(* CoDeSys 2.3.5.6 project: lyjak_02_st.pro *)
(* Author: mgr inż. Tomasz Sklenarski *)
(* Libraries: Standard.lib*4.1.15 17:23:13, SYSLIBCALLBACK.LIB*4.1.15 17:23:13 *)

(* PLC configuration (modules and I/O channels)
I1 AT %IX0.0 [LocalBitInput] Input I1
I2 AT %IX0.1 [LocalBitInput] Input I2
I3 AT %IX0.2 [LocalBitInput] Input I3
I4 AT %IX0.3 [LocalBitInput] Input I4
I5 AT %IX0.4 [LocalBitInput] Input I5
I6 AT %IX0.5 [LocalBitInput] Input I6
I7 AT %IX0.6 [LocalBitInput] Input I7
I8 AT %IX0.7 [LocalBitInput] Input I8
I9 AT %IX1.0 [LocalBitInput] Input I9
I10 AT %IX1.1 [LocalBitInput] Input I10
I11 AT %IX1.2 [LocalBitInput] Input I11
I12 AT %IX1.3 [LocalBitInput] Input I12
I13 AT %IX1.4 [LocalDiagInput] Diagnostic Input I13
I14 AT %IX1.5 [LocalDiagInput] Diagnostic Input I14
I15 AT %IX1.6 [LocalDiagInput] Diagnostic Input I15
I16 AT %IX1.7 [LocalDiagInput] Diagnostic Input I16
I7_Analog AT %IW2 [LocalAnalogIn] Input I7, 10Bit, 0-10VDC
I8_Analog AT %IW4 [LocalAnalogIn] Input I8, 10Bit, 0-10VDC
I11_Analog AT %IW6 [LocalAnalogIn] Input I11, 10Bit, 0-10VDC
I12_Analog AT %IW8 [LocalAnalogIn] Input I12, 10Bit, 0-10VDC
Q1 AT %QX0.0 [LocalBitOutput] Transistor-Output Q1
Q2 AT %QX0.1 [LocalBitOutput] Transistor-Output Q2
Q3 AT %QX0.2 [LocalBitOutput] Transistor-Output Q3
Q4 AT %QX0.3 [LocalBitOutput] Transistor-Output Q4
Q5 AT %QX0.4 [LocalBitOutput] Transistor-Output Q5
Q6 AT %QX0.5 [LocalBitOutput] Transistor-Output Q6
Q7 AT %QX0.6 [LocalBitOutput] Transistor-Output Q7
Q8 AT %QX0.7 [LocalBitOutput] Transistor-Output Q8
No Analog Output [EC4P_NoAnalogOutput] node 1, in %IB10 out %QB1
No Keys [EC4P_NoKeys] node 2, in %IB10 out %QB1
No Counter [EC4P_NoCounter] node 3, in %IB10 out %QB1
Extension [EC4P_Extension] node 1, in %IB10 out %QB1
  No Extension [EC4P_NoExtension] node 0, in %IB10 out %QB1
*)

(* Global variable list: ilosc_bitow_porownania *)
VAR_GLOBAL CONSTANT
	MaxNoOfStates: UINT:=26;
END_VAR

(* Global variable list: wizualizacja *)
VAR_GLOBAL
	numerStanuIn1:BYTE;
	numerStanuIn2:BYTE;
END_VAR

(* Global variable list: ZMIENNE_WYMIANY *)
VAR_GLOBAL
	sterowanieQ12:dataExchange;
	sterowanieQ34:dataExchange;
END_VAR

(* Data type *)
TYPE dataExchange :
STRUCT
	InputState:ARRAY[0..MaxNoOfStates]OF signal;
	Qa:ARRAY[0..MaxNoOfStates]OF signal;
	Qb:ARRAY[0..MaxNoOfStates]OF signal;
END_STRUCT
END_TYPE

(* Data type *)
TYPE signal: (e0, e1, eXX);
END_TYPE

(* POU PLC_PRG, ST *)
PROGRAM PLC_PRG
VAR

	firstRun:BOOL;
	scanner1: scan;
	scan1No:BYTE;
	scanner2: scan;
	scan2No:BYTE;
END_VAR
IF NOT firstRun THEN
i1_config;
i2_config;
firstRun:=TRUE;
END_IF
scanner1(DigIn:=I1 , sigDef:=ADR(sterowanieQ12) , QA=>Q1 , QB=>Q2, No=> numerStanuIn1 );
scanner2(DigIn:=I1 , sigDef:=ADR(sterowanieQ34) , QA=>Q3 , QB=>Q4, No=> numerStanuIn2);
END_PROGRAM
ACTION i1_config:
sterowanieQ12.InputState[2]:=e1;
sterowanieQ12.InputState[3]:=e1;
sterowanieQ12.InputState[4]:=e1;
sterowanieQ12.InputState[5]:=e1;
sterowanieQ12.InputState[6]:=e1;
sterowanieQ12.InputState[7]:=e1;
sterowanieQ12.InputState[8]:=e1;
sterowanieQ12.InputState[9]:=eXX;
sterowanieQ12.InputState[10]:=eXX;
sterowanieQ12.InputState[11]:=e1;
sterowanieQ12.InputState[12]:=e1;

sterowanieQ12.Qa[5]:=e1;
sterowanieQ12.Qa[6]:=e1;
sterowanieQ12.Qa[7]:=e1;
(*
sterowanieQ12.Qa[9]:=eXX;
sterowanieQ12.Qa[10]:=eXX;
*)
sterowanieQ12.Qa[14]:=e1;
sterowanieQ12.Qa[15]:=e1;
sterowanieQ12.Qa[16]:=e1;


sterowanieQ12.Qb[2]:=e1;
sterowanieQ12.Qb[3]:=e1;
sterowanieQ12.Qb[5]:=e1;
sterowanieQ12.Qb[6]:=e1;
(*
sterowanieQ12.Qb[9]:=eXX;
sterowanieQ12.Qb[10]:=eXX;
*)
sterowanieQ12.Qb[17]:=e1;
sterowanieQ12.Qb[18]:=e1;
sterowanieQ12.Qb[21]:=e1;
sterowanieQ12.Qb[22]:=e1;
END_ACTION
ACTION i2_config:
sterowanieQ34.InputState[2]:=e1;
sterowanieQ34.InputState[3]:=e1;
sterowanieQ34.InputState[4]:=e1;
sterowanieQ34.InputState[5]:=e1;
sterowanieQ34.InputState[6]:=e1;
sterowanieQ34.InputState[7]:=e1;
sterowanieQ34.InputState[8]:=e1;
sterowanieQ34.InputState[9]:=e1;
sterowanieQ34.InputState[10]:=e1;
sterowanieQ34.InputState[11]:=eXX;
sterowanieQ34.InputState[12]:=eXX;
sterowanieQ34.InputState[13]:=e1;
sterowanieQ34.InputState[14]:=e1;
sterowanieQ34.InputState[15]:=e1;
sterowanieQ34.InputState[16]:=e1;

sterowanieQ34.Qa[4]:=e1;
sterowanieQ34.Qa[5]:=e1;
sterowanieQ34.Qa[8]:=e1;
sterowanieQ34.Qa[9]:=e1;
sterowanieQ34.Qa[17]:=e1;
sterowanieQ34.Qa[18]:=e1;
sterowanieQ34.Qa[21]:=e1;
sterowanieQ34.Qa[22]:=e1;

sterowanieQ34.Qb[2]:=e1;
sterowanieQ34.Qb[3]:=e1;
sterowanieQ34.Qb[4]:=e1;
sterowanieQ34.Qb[19]:=e1;
sterowanieQ34.Qb[20]:=e1;
END_ACTION

(* POU scan, ST *)
FUNCTION_BLOCK scan
VAR_INPUT
	DigIn:BOOL;
	sigDef:POINTER TO dataExchange;
END_VAR
VAR_OUTPUT
	QA:BOOL;
	QB:BOOL;
	No:BYTE;
END_VAR
VAR
	tim: TON;
	StateMachine:BYTE;
	StateTime:TIME:=t#1s;
END_VAR
CASE StateMachine
OF
0:
IF DigIn THEN
REPEAT
No:=No+1;
UNTIL sigDef^.InputState[No]=e0
END_REPEAT
No:=No+1;
StateMachine:=1;
END_IF
1:
IF tim.Q THEN

IF NOT DigIn AND sigDef^.InputState[No]=eXX THEN
StateMachine:=2;
END_IF
END_IF
2:
StateTime:=t#2s;
IF tim.Q THEN
StateMachine:=3;
StateTime:=t#1s;
END_IF
3:
IF DigIn THEN
StateMachine:=1;
END_IF
END_CASE


tim(IN:=(StateMachine=1 OR StateMachine=2 OR StateMachine=4) AND NOT tim.Q , PT:=StateTime , Q=> , ET=> );
IF tim.Q THEN
No:=No+1;
END_IF
IF No>=MaxNoOfStates THEN
No:=UINT_TO_BYTE(MaxNoOfStates);
END_IF


QA:=sigToBOOL(sigDef^.Qa[No]);
QB:=sigToBOOL(sigDef^.Qb[No]);
END_FUNCTION_BLOCK

(* POU sigToBOOL, ST *)
FUNCTION sigToBOOL : BOOL
VAR_INPUT
	sigIn:signal;
END_VAR
VAR
END_VAR
IF sigIN=e1 THEN
sigToBOOL:=TRUE;
ELSE
sigToBOOL:=FALSE;
END_IF
END_FUNCTION
